Fanuc KAREL source: tst_sim_tof.kl

PROGRAM tst_sim_tof
%NOLOCKGROUP
%UNINITVARS

VAR
  feed_delay FROM test_tof : INTEGER
  sim_file FROM test_tof : STRING[16]
  fl : FILE
  b : BOOLEAN
  val : ARRAY[1] OF REAL
  uninit_r : ARRAY[1] OF REAL
  status : INTEGER
  head : STRING[6]

--port types
%include kliotyps.kl

--sensor definition
%include sensor_calib_test_settings.klt

%from csv.klh %import read_open, read_close, read_line, read_rarr


BEGIN
  --make simulated
  SET_PORT_SIM(io_anin, SENSOR_PIN, 0, status)

  --open csv file
  csv__read_open(sim_file, fl)
  --read header
  head = csv__read_line(sim_file, fl)

  val[1] = 0
  REPEAT
    --read next simulated value
    b = csv__read_rarr(sim_file, fl, ',', val, uninit_r)
    IF b THEN
      --set value
      SET_PORT_VAL(io_anin, SENSOR_PIN, TRUNC(val[1]), status)
    ENDIF
    DELAY feed_delay
  UNTIL(NOT b)

  csv__read_close(fl)

  --unsimulate
  CLR_PORT_SIM(io_anin, SENSOR_PIN, status)

  WRITE TPDISPLAY('AI sim finished!',CR)

END tst_sim_tof
